# EPICS StreamDevice protocol: Gr4-GaussIoc/GaussIoc/ioc_gaussApp/Db/gauss.proto
OutTerminator = LF;
ReadTimeout = 2000;
ReplyTimeout =20000;
resetBuffer {
 out "FETCh:BUFFer:CLear"
}

getModel{

    out"*IDN?";
    in "%37c";
    ExtraInput= Ignore;
}
getXValue{
    out "FETCh:DC? X";
    in "%6f";
    ExtraInput= Ignore;
}
getYValue{
    out "FETCh:DC? Y";
    in "%6f";
    ExtraInput= Ignore;
}
getZValue{
    out "FETCh:DC? Z";
    in "%6f";
    ExtraInput= Ignore;
}
getAllValue{
    out "FETCh:DC? ALL";
    in "%6f";
    ExtraInput= Ignore;
}
